{attribute 'pack_mode' := '1'}
    {attribute 'OPC.UA.DA' := '1'}
    {attribute 'OPC.UA.DA.StructuredType' := '1'}
    (*
    ST_RW_Plc_Device_Status_HMI_IgnitionExp
    ==================================================
    Generated from Ignition UDT: RW_PLC_Device_Status
    Total tags: 3
    Generated on: 2025-09-16 11:33:46
    *)
    TYPE ST_RW_Plc_Device_Status_HMI_IgnitionExp :
    STRUCT
        {attribute 'OPC.UA.DA' := '1'}
        {attribute 'OPC.UA.DA.Access' := '1'}
        Name : STRING := '';		// Read-only tag
        {attribute 'OPC.UA.DA' := '1'}
        {attribute 'OPC.UA.DA.Access' := '1'}
        IPAddress : STRING := '';		// Read-only tag
        {attribute 'OPC.UA.DA' := '1'}
        {attribute 'OPC.UA.DA.Access' := '1'}
        State : DINT := 0;		// Read-only tag
    END_STRUCT
    END_TYPE

(* stored: Version 1.1.0.1
   DUT ST_RW_Plc_Device_Status_HMI_IgnitionExp: Id {84cc13a5-abf2-4e32-9fee-02b5639135d5} *)
